// TIA Portal V19 program export: 1 tag tables, 1 data types, 3 data blocks, 18 code blocks (in call order from the OBs), 11 instance data blocks

VAR_GLOBAL   // PLC tag table "Default tag table"
   System_Byte AT %MB1 : Byte;
   FirstScan AT %M1.0 : Bool;
   DiagStatusUpdate AT %M1.1 : Bool;
   AlwaysTRUE AT %M1.2 : Bool;
   AlwaysFALSE AT %M1.3 : Bool;
   Clock_Byte AT %MB0 : Byte;
   Clock_10Hz AT %M0.0 : Bool;
   Clock_5Hz AT %M0.1 : Bool;
   "Clock_2.5Hz" AT %M0.2 : Bool;
   Clock_2Hz AT %M0.3 : Bool;
   "Clock_1.25Hz" AT %M0.4 : Bool;
   Clock_1Hz AT %M0.5 : Bool;
   "Clock_0.625Hz" AT %M0.6 : Bool;
   "Clock_0.5Hz" AT %M0.7 : Bool;
   Emergency_Stop_OK AT %M52.2 : Bool;   // Emergency status. 0 = OK, 1 = Emergency
   Emergency_Stop_Status_150K1 AT %I1.0 : Bool;   // Emergency signal from 150K1
   Sensor_102B2 AT %I1.1 : Bool;   // Sensor on conveyor - Front
   Sensor_102B3 AT %I1.2 : Bool;   // Sensor on conveyor - Middle
   Sensor_102B4 AT %I1.3 : Bool;   // Sensor on conveyor - Back
   Sensor_102B5 AT %I1.4 : Bool;   // Paint level sensor - High
   Sensor_102B6 AT %I1.5 : Bool;   // Paint level sensor - Low
   Valve_106Q6 AT %Q1.0 : Bool;   // Paint dispenser valve
   Motor_4Q3 AT %Q1.1 : Bool;   // Contactor for motor - Grinder
   Motor_4Q5 AT %Q1.2 : Bool;   // Contactor for motor - Paint
   Motor_6Q1 AT %Q1.3 : Bool;   // Contactor for motor - Ventilation
   Motor_6Q3 AT %Q1.4 : Bool;   // Contactor for motor - Vacuum
   Reset_Safety_150K1 AT %Q1.5 : Bool;   // Signal to 150K1 for emergency reset
   HMI_Start AT %M51.6 : Bool;   // HMI button signal - Start
   HMI_Pause AT %M51.7 : Bool;   // HMI button signal - Pause
   HMI_Reset AT %M52.0 : Bool;   // HMI button signal - Reset
   Input0 AT %I0.0 : Bool;
   Input1 AT %I0.1 : Bool;
   Input2 AT %I0.2 : Bool;
   Input3 AT %I0.3 : Bool;
   Input4 AT %I0.4 : Bool;
   Input5 AT %I0.5 : Bool;
   Input6 AT %I0.6 : Bool;
   Input7 AT %I0.7 : Bool;
   Input8 AT %I1.6 : Bool;
   Output0 AT %Q0.0 : Bool;
   Output1 AT %Q0.1 : Bool;
   Output2 AT %Q0.2 : Bool;
   Output3 AT %Q0.3 : Bool;
   Output4 AT %Q0.4 : Bool;
   Output5 AT %Q0.5 : Bool;
   Output6 AT %Q0.6 : Bool;
   Output7 AT %Q0.7 : Bool;
   Output8 AT %Q1.6 : Bool;
END_VAR

TYPE "XYZ_Coordinates"
   STRUCT
      X : Int;
      Y : Int;
      Z : Int;
      Mode : Int;
   END_STRUCT;
END_TYPE

DATA_BLOCK "DB_Arduino_Data"   // DB3
{ S7_Optimized_Access := 'FALSE' }
   VAR
      Read_Data : Array[1..120] of Word;
      Write_Data : Array[1..120] of Word;
   END_VAR
BEGIN
   Write_Data[1] := 16#B;
   Write_Data[2] := 16#E;
   Write_Data[3] := 16#0;
END_DATA_BLOCK

DATA_BLOCK "DB_Arduino_Tcp_Connect"   // DB10
{ S7_Optimized_Access := 'TRUE' }
// stored: MemoryReserve 100
   VAR
      MB_Arduino_Write : TCON_IP_v4;
      MB_Arduino_Read : TCON_IP_v4;
      MB_Arduino_Disconnect { S7_SetPoint := 'True'} : Bool;
      MB_Arduino_Req : Bool;
      MB_Arduino_Error : Bool;
      MB_Arduino_Done : Bool;
      MB_Arduino_Busy : Bool;
      MB_Arduino_Status : Word;
      MB_Arduino_Write_Busy : Bool;
      MB_Arduino_Write_Done : Bool;
      MB_Arduino_Write_Error : Bool;
      MB_Arduino_Write_Req : Bool;
      MB_Arduino_Write_Disconnect : Bool;
      MB_Arduino_Write_Status : Word;
   END_VAR
BEGIN
   MB_Arduino_Write.InterfaceId := 64;
   MB_Arduino_Write.ID := 16#1;
   MB_Arduino_Write.ConnectionType := 16#0B;
   MB_Arduino_Write.ActiveEstablished := 1;
   MB_Arduino_Write.RemoteAddress.ADDR[1] := 16#C0;
   MB_Arduino_Write.RemoteAddress.ADDR[2] := 16#A8;
   MB_Arduino_Write.RemoteAddress.ADDR[3] := 16#1;
   MB_Arduino_Write.RemoteAddress.ADDR[4] := 16#3D;
   MB_Arduino_Write.RemotePort := 502;
   MB_Arduino_Read.InterfaceId := 64;
   MB_Arduino_Read.ID := 16#1;
   MB_Arduino_Read.ConnectionType := 16#0B;
   MB_Arduino_Read.ActiveEstablished := 1;
   MB_Arduino_Read.RemoteAddress.ADDR[1] := 16#C0;
   MB_Arduino_Read.RemoteAddress.ADDR[2] := 16#A8;
   MB_Arduino_Read.RemoteAddress.ADDR[3] := 16#1;
   MB_Arduino_Read.RemoteAddress.ADDR[4] := 16#3D;
   MB_Arduino_Read.RemotePort := 502;
END_DATA_BLOCK

DATA_BLOCK "Letter_A"   // DB4
{ S7_Optimized_Access := 'TRUE' }
// stored: MemoryReserve 100
   VAR
      Coordinates : Array[0..5] of "XYZ_Coordinates";
   END_VAR
BEGIN
   Coordinates[0..2].X := 1.0;
   Coordinates[0..2].Y := 2.0;
   Coordinates[0..2].Z := 3.0;
END_DATA_BLOCK

ORGANIZATION_BLOCK "Main"   // OB1, LAD, ProgramCycle
TITLE = "Main Program Sweep (Cycle)"
{ S7_Optimized_Access := 'TRUE' }
// stored: SetENOAutomatically false
   VAR_INPUT
      Initial_Call : Bool;   // Initial call of this OB
      Remanence : Bool;   // =True, if remanent data are available
   END_VAR
   VAR_TEMP   // added for the SCL form of the ladder/FBD networks
      _w1 : Bool;
   END_VAR
BEGIN

REGION Network 1
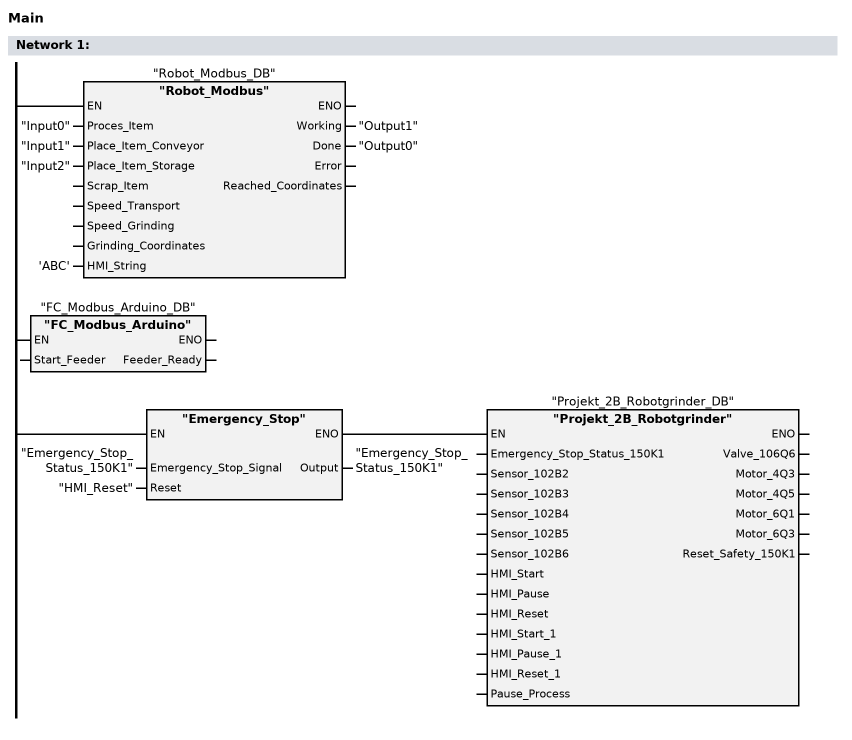
   RUNG wire#powerrail
      "Robot_Modbus_DB"(Proces_Item := "Input0", Place_Item_Conveyor := "Input1", Place_Item_Storage := "Input2", Scrap_Item :=, Speed_Transport :=, Speed_Grinding :=, Grinding_Coordinates :=, HMI_String := 'ABC', Working => "Output1", Done => "Output0", Error =>, Reached_Coordinates =>)
   END_RUNG
   RUNG wire#powerrail
      "FC_Modbus_Arduino_DB"(Start_Feeder :=, Feeder_Ready =>)
   END_RUNG
   RUNG wire#powerrail
      "Emergency_Stop"(Emergency_Stop_Signal := "Emergency_Stop_Status_150K1", Reset := "HMI_Reset", Output => "Emergency_Stop_Status_150K1")
      "Projekt_2B_Robotgrinder_DB"(Emergency_Stop_Status_150K1 :=, Sensor_102B2 :=, Sensor_102B3 :=, Sensor_102B4 :=, Sensor_102B5 :=, Sensor_102B6 :=, HMI_Start :=, HMI_Pause :=, HMI_Reset :=, HMI_Start_1 :=, HMI_Pause_1 :=, HMI_Reset_1 :=, Pause_Process :=, Valve_106Q6 =>, Motor_4Q3 =>, Motor_4Q5 =>, Motor_6Q1 =>, Motor_6Q3 =>, Reset_Safety_150K1 =>)
   END_RUNG
   // the same network as SCL:
   "Robot_Modbus_DB"(Proces_Item := "Input0",   // "Robot_Modbus"
                     Place_Item_Conveyor := "Input1",
                     Place_Item_Storage := "Input2",
                     HMI_String := 'ABC',
                     Working => "Output1",
                     Done => "Output0");
   "FC_Modbus_Arduino_DB"();   // "FC_Modbus_Arduino"
   "Emergency_Stop"(Emergency_Stop_Signal := "Emergency_Stop_Status_150K1",
                    Reset := "HMI_Reset",
                    Output => "Emergency_Stop_Status_150K1",
                    ENO => #_w1);
   IF #_w1 THEN
       "Projekt_2B_Robotgrinder_DB"();   // "Projekt_2B_Robotgrinder"
   END_IF;
END_REGION
END_ORGANIZATION_BLOCK

FUNCTION_BLOCK "Robot_Modbus"   // FB1, LAD
{ S7_Optimized_Access := 'TRUE' }
// V.0.1.1 - Updated UR robot array address
// V.0.1.0 - Created function block
// stored: MemoryReserve 100, SetENOAutomatically false
   VAR_INPUT
      Proces_Item : Bool;
      Place_Item_Conveyor : Bool;
      Place_Item_Storage : Bool;
      Scrap_Item : Bool;
      Speed_Transport : Int := 10;
      Speed_Grinding : Int := 10;
      Grinding_Coordinates : Bool;
      HMI_String : String;
   END_VAR
   VAR_OUTPUT
      Working : Bool;
      Done : Bool;
      Error : Bool;
      Reached_Coordinates : Bool;
   END_VAR
   VAR
      DISCONNECT : Bool;
      Address : TCON_IP_v4;
      Receive_Data : Int;
      Send_Data : Array[0..63] of Bool;
      Send_Coordinates : Array[0..2] of Int;
      Letter_A : Array[0..20] of "XYZ_Coordinates";
      Letter_Steps { S7_SetPoint := 'True'} : Int;
      Rising_edge : Bool;
      String_To_Letter_Array : Array[0..16] of Char;
      String_Length : Int;
      Currently_Processing : Int;
      Send_Letter_A : Bool;
      Send_Letter_B : Bool;
      Send_Letter_C : Bool;
      MB_Client_Mode : Int;
      MB_Client_Modbus_Address : Int;
      For_Loop_Counter : Int;
   END_VAR
   // Address.InterfaceId := 64;
   // Address.ID := 1;
   // Address.ConnectionType := 11;
   // Address.ActiveEstablished := TRUE;
   // Address.RemoteAddress.ADDR[1] := 192;
   // Address.RemoteAddress.ADDR[2] := 168;
   // Address.RemoteAddress.ADDR[3] := 1;
   // Address.RemoteAddress.ADDR[4] := 51;
   // Address.RemotePort := 502;
   // Address.LocalPort := 502;
   // Letter_A[0..1].X := 4;
   // Letter_A[2].X := 42;
   // Letter_A[3].X := 56;
   // Letter_A[4].X := 98;
   // Letter_A[5].X := 82;
   // Letter_A[6].X := 70;
   // Letter_A[7].X := 29;
   // Letter_A[8].X := 17;
   // Letter_A[9..10].X := 4;
   // Letter_A[11..12].X := 67;
   // Letter_A[13].X := 56;
   // Letter_A[14].X := 52;
   // Letter_A[15].X := 49;
   // Letter_A[16].X := 47;
   // Letter_A[17].X := 44;
   // Letter_A[18..19].X := 33;
   // Letter_A[0].Y := 0;
   // Letter_A[2..3].Y := 100;
   // Letter_A[4..5].Y := 0;
   // Letter_A[6..7].Y := 30;
   // Letter_A[8..10].Y := 0;
   // Letter_A[11..12].Y := 41;
   // Letter_A[13].Y := 69;
   // Letter_A[14].Y := 82;
   // Letter_A[15].Y := 90;
   // Letter_A[16].Y := 80;
   // Letter_A[17].Y := 70;
   // Letter_A[18..19].Y := 41;
   // Letter_A[1..9].Z := -1;
   // Letter_A[10].Z := 0;
   // Letter_A[12..18].Z := -1;
   // Letter_A[19].Z := 0;
   // Letter_A[14].I := 394;
   // Letter_A[15].I := 156;
   // Letter_A[16].I := -122;
   // Letter_A[17].I := -127;
   // Letter_A[14].J := 149;
   // Letter_A[15].J := 53;
   // Letter_A[16].J := 24;
   // Letter_A[17].J := 36;
   VAR_TEMP   // added for the SCL form of the ladder/FBD networks
      _w1 : Bool;
   END_VAR
BEGIN

REGION Network 1: MB_CLIENT
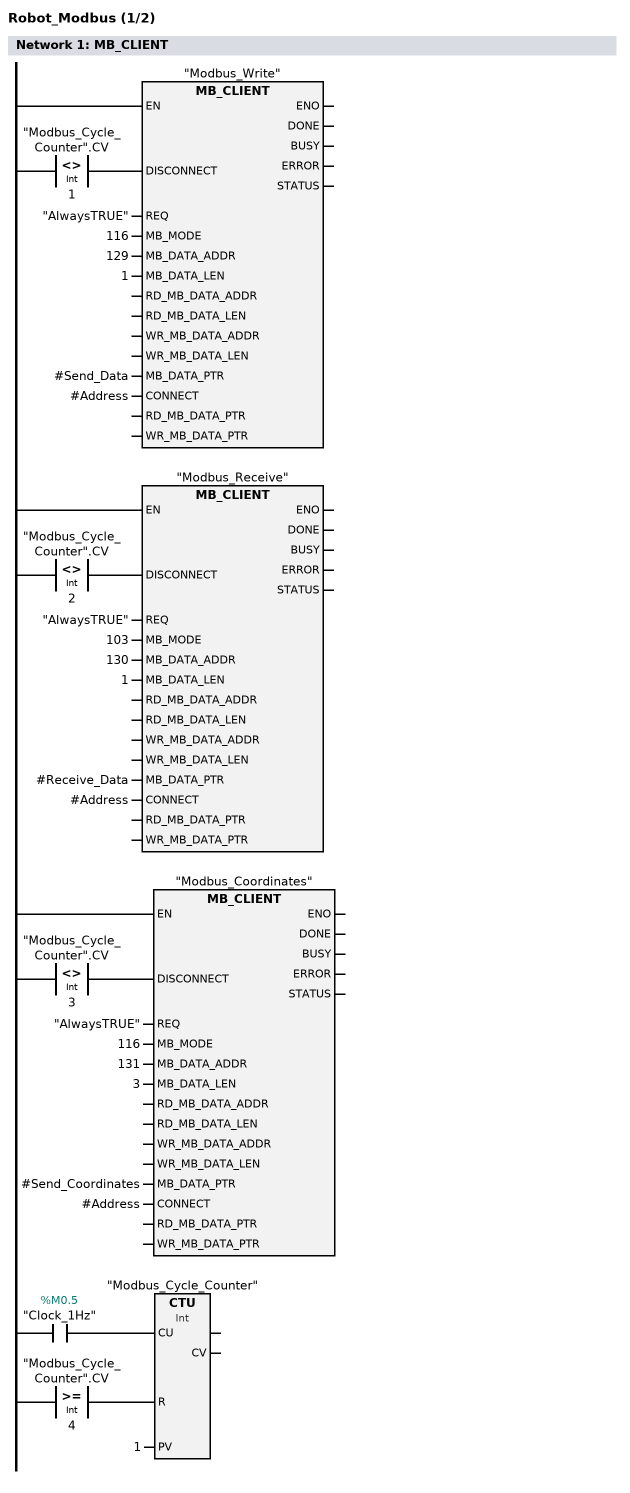
   RUNG wire#powerrail
      "Modbus_Write".MB_CLIENT(DISCONNECT := wire#w1, REQ := "AlwaysTRUE", MB_MODE := 116, MB_DATA_ADDR := 129, MB_DATA_LEN := 1, RD_MB_DATA_ADDR :=, RD_MB_DATA_LEN :=, WR_MB_DATA_ADDR :=, WR_MB_DATA_LEN :=, MB_DATA_PTR := #Send_Data, CONNECT := #Address, RD_MB_DATA_PTR :=, WR_MB_DATA_PTR :=, DONE =>, BUSY =>, ERROR =>, STATUS =>)
   END_RUNG
   RUNG wire#powerrail
      { S7_Templates := "SrcType := Int" } NE_Contact(in1 := "Modbus_Cycle_Counter".CV, in2 := 1)
   END_RUNG wire#w1
   RUNG wire#powerrail
      "Modbus_Receive".MB_CLIENT(DISCONNECT := wire#w2, REQ := "AlwaysTRUE", MB_MODE := 103, MB_DATA_ADDR := 130, MB_DATA_LEN := 1, RD_MB_DATA_ADDR :=, RD_MB_DATA_LEN :=, WR_MB_DATA_ADDR :=, WR_MB_DATA_LEN :=, MB_DATA_PTR := #Receive_Data, CONNECT := #Address, RD_MB_DATA_PTR :=, WR_MB_DATA_PTR :=, DONE =>, BUSY =>, ERROR =>, STATUS =>)
   END_RUNG
   RUNG wire#powerrail
      { S7_Templates := "SrcType := Int" } NE_Contact(in1 := "Modbus_Cycle_Counter".CV, in2 := 2)
   END_RUNG wire#w2
   RUNG wire#powerrail
      "Modbus_Coordinates".MB_CLIENT(DISCONNECT := wire#w3, REQ := "AlwaysTRUE", MB_MODE := 116, MB_DATA_ADDR := 131, MB_DATA_LEN := 3, RD_MB_DATA_ADDR :=, RD_MB_DATA_LEN :=, WR_MB_DATA_ADDR :=, WR_MB_DATA_LEN :=, MB_DATA_PTR := #Send_Coordinates, CONNECT := #Address, RD_MB_DATA_PTR :=, WR_MB_DATA_PTR :=, DONE =>, BUSY =>, ERROR =>, STATUS =>)
   END_RUNG
   RUNG wire#powerrail
      { S7_Templates := "SrcType := Int" } NE_Contact(in1 := "Modbus_Cycle_Counter".CV, in2 := 3)
   END_RUNG wire#w3
   RUNG wire#powerrail
      Contact( "Clock_1Hz" )
      { S7_Templates := "value_type := Int" } "Modbus_Cycle_Counter".CTU(r := wire#w4, pv := 1, cv =>)
   END_RUNG
   RUNG wire#powerrail
      { S7_Templates := "SrcType := Int" } GE_Contact(in1 := "Modbus_Cycle_Counter".CV, in2 := 4)
   END_RUNG wire#w4
   // the same network as SCL:
   "Modbus_Write"(DISCONNECT := "Modbus_Cycle_Counter".CV <> 1,   // MB_CLIENT
                  REQ := "AlwaysTRUE",
                  MB_MODE := 116,
                  MB_DATA_ADDR := 129,
                  MB_DATA_LEN := 1,
                  MB_DATA_PTR := #Send_Data,
                  CONNECT := #Address);
   "Modbus_Receive"(DISCONNECT := "Modbus_Cycle_Counter".CV <> 2,   // MB_CLIENT
                    REQ := "AlwaysTRUE",
                    MB_MODE := 103,
                    MB_DATA_ADDR := 130,
                    MB_DATA_LEN := 1,
                    MB_DATA_PTR := #Receive_Data,
                    CONNECT := #Address);
   "Modbus_Coordinates"(DISCONNECT := "Modbus_Cycle_Counter".CV <> 3,   // MB_CLIENT
                        REQ := "AlwaysTRUE",
                        MB_MODE := 116,
                        MB_DATA_ADDR := 131,
                        MB_DATA_LEN := 3,
                        MB_DATA_PTR := #Send_Coordinates,
                        CONNECT := #Address);
   "Modbus_Cycle_Counter".CTU(CU := "Clock_1Hz", R := "Modbus_Cycle_Counter".CV >= 4, PV := 1);
END_REGION

REGION Network 2: Send Data
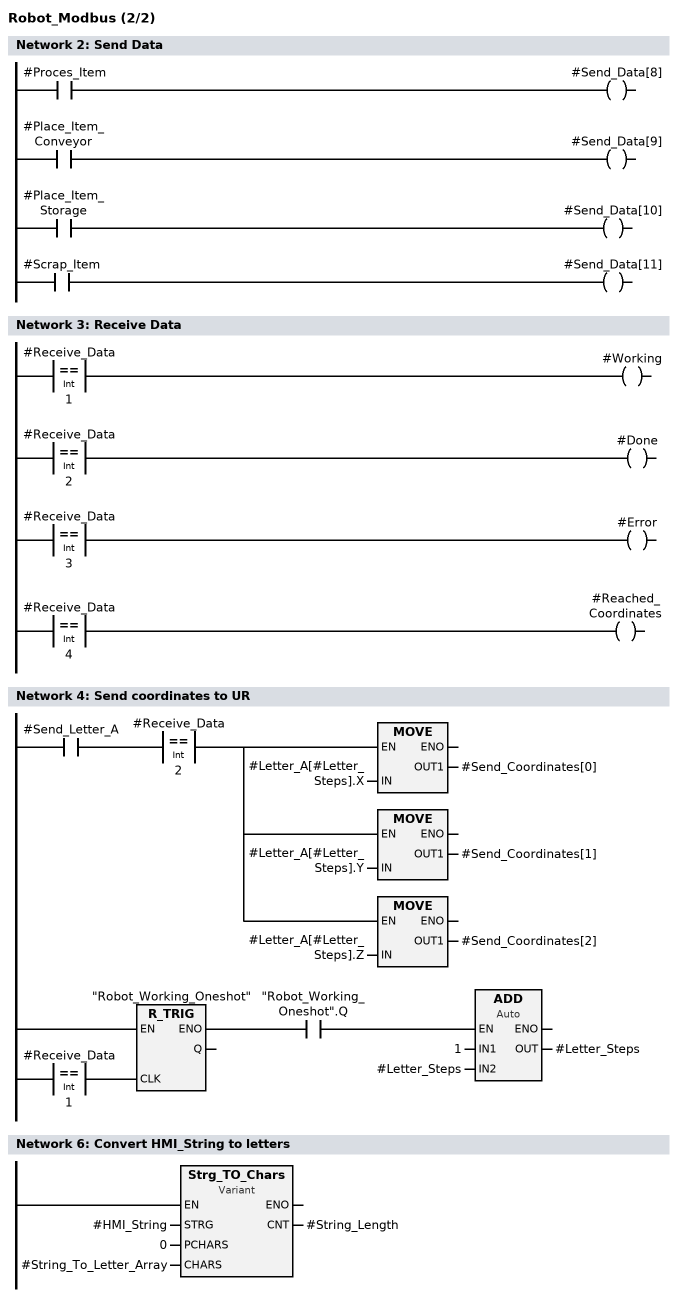
   RUNG wire#powerrail
      Contact( #Proces_Item )
      Coil( #Send_Data[8] )
   END_RUNG
   RUNG wire#powerrail
      Contact( #Place_Item_Conveyor )
      Coil( #Send_Data[9] )
   END_RUNG
   RUNG wire#powerrail
      Contact( #Place_Item_Storage )
      Coil( #Send_Data[10] )
   END_RUNG
   RUNG wire#powerrail
      Contact( #Scrap_Item )
      Coil( #Send_Data[11] )
   END_RUNG
   // the same network as SCL:
   #Send_Data[8] := #Proces_Item;
   #Send_Data[9] := #Place_Item_Conveyor;
   #Send_Data[10] := #Place_Item_Storage;
   #Send_Data[11] := #Scrap_Item;
END_REGION

REGION Network 3: Receive Data
   RUNG wire#powerrail
      { S7_Templates := "SrcType := Int" } EQ_Contact(in1 := #Receive_Data, in2 := 1)
      Coil( #Working )
   END_RUNG
   RUNG wire#powerrail
      { S7_Templates := "SrcType := Int" } EQ_Contact(in1 := #Receive_Data, in2 := 2)
      Coil( #Done )
   END_RUNG
   RUNG wire#powerrail
      { S7_Templates := "SrcType := Int" } EQ_Contact(in1 := #Receive_Data, in2 := 3)
      Coil( #Error )
   END_RUNG
   RUNG wire#powerrail
      { S7_Templates := "SrcType := Int" } EQ_Contact(in1 := #Receive_Data, in2 := 4)
      Coil( #Reached_Coordinates )
   END_RUNG
   // the same network as SCL:
   #Working := #Receive_Data = 1;
   #Done := #Receive_Data = 2;
   #Error := #Receive_Data = 3;
   #Reached_Coordinates := #Receive_Data = 4;
END_REGION

REGION Network 4: Send coordinates to UR
   RUNG wire#powerrail
      Contact( #Send_Letter_A )
      { S7_Templates := "SrcType := Int" } EQ_Contact(in1 := #Receive_Data, in2 := 2)
      wire#w1
      Move(in := #Letter_A[#Letter_Steps].X, out1 => #Send_Coordinates[0])
   END_RUNG
   RUNG wire#w1
      Move(in := #Letter_A[#Letter_Steps].Y, out1 => #Send_Coordinates[1])
   END_RUNG
   RUNG wire#w1
      Move(in := #Letter_A[#Letter_Steps].Z, out1 => #Send_Coordinates[2])
   END_RUNG
   RUNG wire#powerrail
      "Robot_Working_Oneshot".R_TRIG(CLK := wire#w2, Q =>)
      Contact( "Robot_Working_Oneshot".Q )
      Add(in1 := 1, in2 := #Letter_Steps, out => #Letter_Steps)
   END_RUNG
   RUNG wire#powerrail
      { S7_Templates := "SrcType := Int" } EQ_Contact(in1 := #Receive_Data, in2 := 1)
   END_RUNG wire#w2
   // the same network as SCL:
   IF #Send_Letter_A AND (#Receive_Data = 2) THEN
       #Send_Coordinates[0] := #Letter_A[#Letter_Steps].X;
       #Send_Coordinates[1] := #Letter_A[#Letter_Steps].Y;
       #Send_Coordinates[2] := #Letter_A[#Letter_Steps].Z;
   END_IF;
   "Robot_Working_Oneshot"(CLK := #Receive_Data = 1, ENO => #_w1);   // R_TRIG
   IF #_w1 AND "Robot_Working_Oneshot".Q THEN #Letter_Steps := 1 + #Letter_Steps; END_IF;
END_REGION

REGION Network 5 (SCL): Insert coordinates into Modbus_Data array
   (*
   //If we need to make letter A, and robot is sending ready signal
   IF #Send_Letter_A AND #Send_Data[25] THEN

       FOR #For_Loop_Counter := 32 TO 48 DO
           //Find the bit state inside to INT of letter_A array, and copy that to the Modbus data array
           //The for loop repeats the steps again for the array posistions 32-48
           #Letter_A[#Letter_Steps].X.%X0 := #Send_Data[#For_Loop_Counter];
       END_FOR;

       FOR #For_Loop_Counter := 49 TO 64 DO
           #Letter_A[#Letter_Steps].Y.%X0 := #Send_Data[#For_Loop_Counter];
       END_FOR;

       FOR #For_Loop_Counter := 65 TO 79 DO
           #Letter_A[#Letter_Steps].Z.%X0 := #Send_Data[#For_Loop_Counter];
       END_FOR;

   END_IF; *)
END_REGION

REGION Network 6: Convert HMI_String to letters
   RUNG wire#powerrail
      { S7_Templates := "[ptr_type := Variant, strg_type := String]" } Strg_TO_Chars(Strg := #HMI_String, pChars := 0, Chars := #String_To_Letter_Array, Cnt => #String_Length)
   END_RUNG
   // the same network as SCL:
   Strg_TO_Chars(Strg := #HMI_String, pChars := 0, Chars := #String_To_Letter_Array, Cnt => #String_Length);
END_REGION

REGION Network 7 (SCL)
   IF #Currently_Processing < #String_Length THEN //Hvis vi ikke er nået forbi enden af teksten

       IF #String_To_Letter_Array[#Currently_Processing] = 'A' THEN //Hvis der på position X, er et "A" i teksten
           #Send_Letter_A := TRUE;
       ELSIF #String_To_Letter_Array[#Currently_Processing] = 'B' THEN
           #Send_Letter_B := TRUE;
       ELSIF #String_To_Letter_Array[#Currently_Processing] = 'C' THEN
           #Send_Letter_B := TRUE;
       END_IF;
   END_IF;
END_REGION
END_FUNCTION_BLOCK

FUNCTION_BLOCK "FC_Modbus_Arduino"   // FB1, LAD
{ S7_Optimized_Access := 'TRUE' }
// stored: MemoryReserve 100, SetENOAutomatically false
   VAR_INPUT
      Start_Feeder : Bool;
   END_VAR
   VAR_OUTPUT
      Feeder_Ready : Bool;
   END_VAR
BEGIN

REGION Network 1
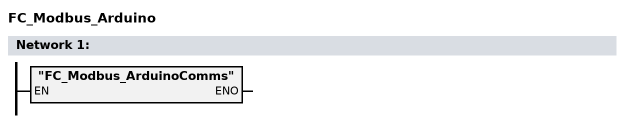
   RUNG wire#powerrail
      "FC_Modbus_ArduinoComms"()
   END_RUNG
   // the same network as SCL:
   "FC_Modbus_ArduinoComms"();
END_REGION
END_FUNCTION_BLOCK

FUNCTION "FC_Modbus_ArduinoComms" : Void   // FC1, LAD
{ S7_Optimized_Access := 'TRUE' }
// stored: SetENOAutomatically false
BEGIN

REGION Network 1
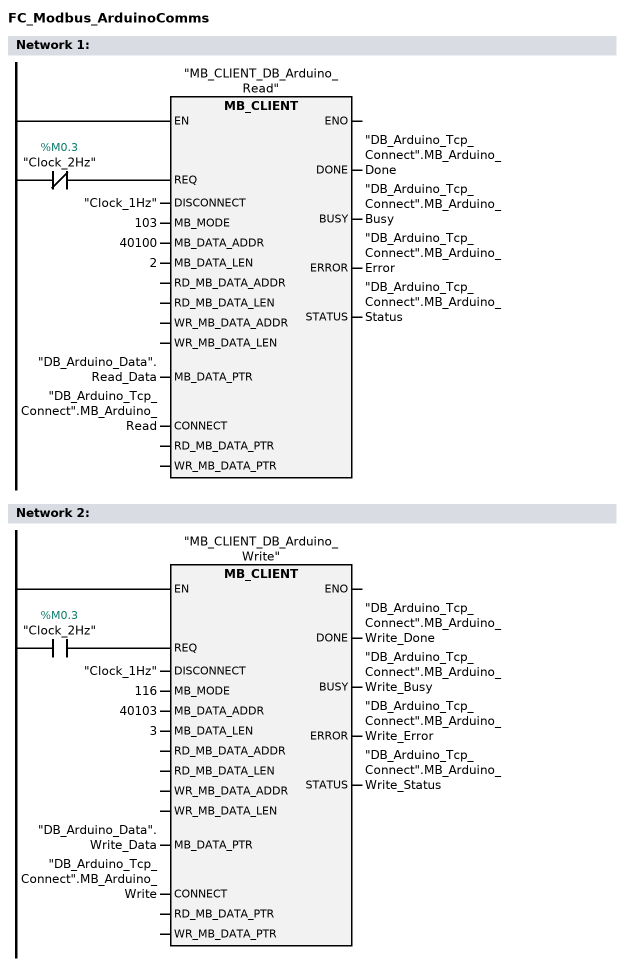
   RUNG wire#powerrail
      "MB_CLIENT_DB_Arduino_Read".MB_CLIENT(REQ := wire#w1, DISCONNECT := "Clock_1Hz", MB_MODE := 103, MB_DATA_ADDR := 40100, MB_DATA_LEN := 2, RD_MB_DATA_ADDR :=, RD_MB_DATA_LEN :=, WR_MB_DATA_ADDR :=, WR_MB_DATA_LEN :=, MB_DATA_PTR := "DB_Arduino_Data".Read_Data, CONNECT := "DB_Arduino_Tcp_Connect".MB_Arduino_Read, RD_MB_DATA_PTR :=, WR_MB_DATA_PTR :=, DONE => "DB_Arduino_Tcp_Connect".MB_Arduino_Done, BUSY => "DB_Arduino_Tcp_Connect".MB_Arduino_Busy, ERROR => "DB_Arduino_Tcp_Connect".MB_Arduino_Error, STATUS => "DB_Arduino_Tcp_Connect".MB_Arduino_Status)
   END_RUNG
   RUNG wire#powerrail
      I_Contact( "Clock_2Hz" )
   END_RUNG wire#w1
   // the same network as SCL:
   "MB_CLIENT_DB_Arduino_Read"(REQ := NOT "Clock_2Hz",   // MB_CLIENT
                           DISCONNECT := "Clock_1Hz",
                           MB_MODE := 103,
                           MB_DATA_ADDR := 40100,
                           MB_DATA_LEN := 2,
                           MB_DATA_PTR := "DB_Arduino_Data".Read_Data,
                           CONNECT := "DB_Arduino_Tcp_Connect".MB_Arduino_Read,
                           DONE => "DB_Arduino_Tcp_Connect".MB_Arduino_Done,
                           BUSY => "DB_Arduino_Tcp_Connect".MB_Arduino_Busy,
                           ERROR => "DB_Arduino_Tcp_Connect".MB_Arduino_Error,
                           STATUS => "DB_Arduino_Tcp_Connect".MB_Arduino_Status);
END_REGION

REGION Network 2
   RUNG wire#powerrail
      "MB_CLIENT_DB_Arduino_Write".MB_CLIENT(REQ := wire#w1, DISCONNECT := "Clock_1Hz", MB_MODE := 116, MB_DATA_ADDR := 40103, MB_DATA_LEN := 3, RD_MB_DATA_ADDR :=, RD_MB_DATA_LEN :=, WR_MB_DATA_ADDR :=, WR_MB_DATA_LEN :=, MB_DATA_PTR := "DB_Arduino_Data".Write_Data, CONNECT := "DB_Arduino_Tcp_Connect".MB_Arduino_Write, RD_MB_DATA_PTR :=, WR_MB_DATA_PTR :=, DONE => "DB_Arduino_Tcp_Connect".MB_Arduino_Write_Done, BUSY => "DB_Arduino_Tcp_Connect".MB_Arduino_Write_Busy, ERROR => "DB_Arduino_Tcp_Connect".MB_Arduino_Write_Error, STATUS => "DB_Arduino_Tcp_Connect".MB_Arduino_Write_Status)
   END_RUNG
   RUNG wire#powerrail
      Contact( "Clock_2Hz" )
   END_RUNG wire#w1
   // the same network as SCL:
   "MB_CLIENT_DB_Arduino_Write"(REQ := "Clock_2Hz",   // MB_CLIENT
                           DISCONNECT := "Clock_1Hz",
                           MB_MODE := 116,
                           MB_DATA_ADDR := 40103,
                           MB_DATA_LEN := 3,
                           MB_DATA_PTR := "DB_Arduino_Data".Write_Data,
                           CONNECT := "DB_Arduino_Tcp_Connect".MB_Arduino_Write,
                           DONE => "DB_Arduino_Tcp_Connect".MB_Arduino_Write_Done,
                           BUSY => "DB_Arduino_Tcp_Connect".MB_Arduino_Write_Busy,
                           ERROR => "DB_Arduino_Tcp_Connect".MB_Arduino_Write_Error,
                           STATUS => "DB_Arduino_Tcp_Connect".MB_Arduino_Write_Status);
END_REGION
END_FUNCTION

FUNCTION "Emergency_Stop" : Void
{ S7_Optimized_Access := 'TRUE' }
VERSION : 0.1
   VAR_INPUT 
      Emergency_Stop_Signal : Bool;
      Reset : Bool;
   END_VAR

   VAR_OUTPUT 
      Output : Bool;
   END_VAR


BEGIN
	IF #Emergency_Stop_Signal = TRUE THEN
	    #Output := TRUE;
	END_IF;
	    
	IF #Reset = TRUE AND #Emergency_Stop_Signal = FALSE THEN
	    #Output := FALSE;
	END_IF;
END_FUNCTION

FUNCTION_BLOCK "Projekt_2B_Robotgrinder"   // FB4, LAD
{ S7_Optimized_Access := 'TRUE' }
// stored: MemoryReserve 100, SetENOAutomatically false
   VAR_INPUT
      Emergency_Stop_Status_150K1 : Bool;
      Sensor_102B2 : Bool;
      Sensor_102B3 : Bool;
      Sensor_102B4 : Bool;
      Sensor_102B5 : Bool;
      Sensor_102B6 : Bool;
      HMI_Start : Bool;
      HMI_Pause : Bool;
      HMI_Reset : Bool;
      HMI_Start_1 : Bool;
      HMI_Pause_1 : Bool;
      HMI_Reset_1 : Bool;
      Pause_Process : Bool;
   END_VAR
   VAR_OUTPUT
      Valve_106Q6 : Bool;
      Motor_4Q3 : Bool;
      Motor_4Q5 : Bool;
      Motor_6Q1 : Bool;
      Motor_6Q3 : Bool;
      Reset_Safety_150K1 : Bool;
   END_VAR
   VAR
      Main_Step : Int;
      Process_Step : Int;
      Reset_Step : Int;
      Placement_Step : Int;
      Order_Amount : Int;
      Items_Produced : Int;
      Items_Delivered : Int;
      Total_orders : Int;
      Storage_Amount : Int;
      Storage_Plus_Produce : Int;
      Storage_Min : Int;
      Storage_Max : Int;
      Robot_Done : Bool;
   END_VAR
BEGIN

REGION Network 1: Main Process Step 0
   // If the system is currently idling, then pressing start will start the process. On PLC restart, moves starting values into steps.
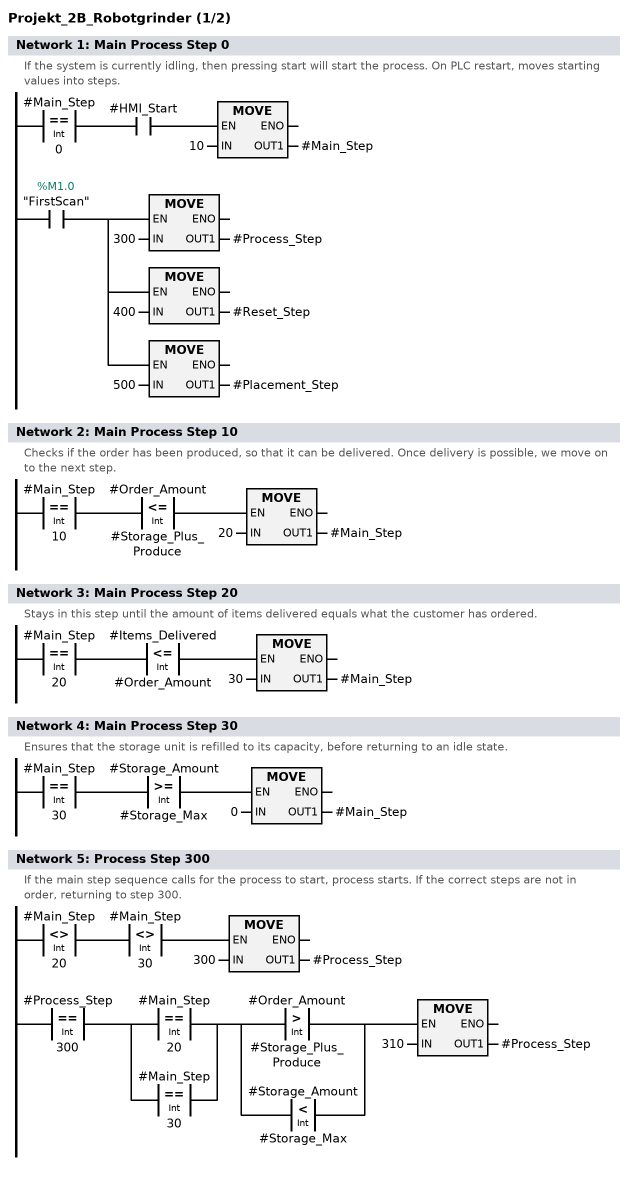
   RUNG wire#powerrail
      { S7_Templates := "SrcType := Int" } EQ_Contact(in1 := #Main_Step, in2 := 0)
      Contact( #HMI_Start )
      Move(in := 10, out1 => #Main_Step)
   END_RUNG
   RUNG wire#powerrail
      Contact( "FirstScan" )
      wire#w1
      Move(in := 300, out1 => #Process_Step)
   END_RUNG
   RUNG wire#w1
      Move(in := 400, out1 => #Reset_Step)
   END_RUNG
   RUNG wire#w1
      Move(in := 500, out1 => #Placement_Step)
   END_RUNG
   // the same network as SCL:
   IF (#Main_Step = 0) AND #HMI_Start THEN #Main_Step := 10; END_IF;
   IF "FirstScan" THEN
       #Process_Step := 300;
       #Reset_Step := 400;
       #Placement_Step := 500;
   END_IF;
END_REGION

REGION Network 2: Main Process Step 10
   // Checks if the order has been produced, so that it can be delivered. Once delivery is possible, we move on to the next step.
   RUNG wire#powerrail
      { S7_Templates := "SrcType := Int" } EQ_Contact(in1 := #Main_Step, in2 := 10)
      { S7_Templates := "SrcType := Int" } LE_Contact(in1 := #Order_Amount, in2 := #Storage_Plus_Produce)
      Move(in := 20, out1 => #Main_Step)
   END_RUNG
   // the same network as SCL:
   IF (#Main_Step = 10) AND (#Order_Amount <= #Storage_Plus_Produce) THEN #Main_Step := 20; END_IF;
END_REGION

REGION Network 3: Main Process Step 20
   // Stays in this step until the amount of items delivered equals what the customer has ordered.
   RUNG wire#powerrail
      { S7_Templates := "SrcType := Int" } EQ_Contact(in1 := #Main_Step, in2 := 20)
      { S7_Templates := "SrcType := Int" } LE_Contact(in1 := #Items_Delivered, in2 := #Order_Amount)
      Move(in := 30, out1 => #Main_Step)
   END_RUNG
   // the same network as SCL:
   IF (#Main_Step = 20) AND (#Items_Delivered <= #Order_Amount) THEN #Main_Step := 30; END_IF;
END_REGION

REGION Network 4: Main Process Step 30
   // Ensures that the storage unit is refilled to its capacity, before returning to an idle state.
   RUNG wire#powerrail
      { S7_Templates := "SrcType := Int" } EQ_Contact(in1 := #Main_Step, in2 := 30)
      { S7_Templates := "SrcType := Int" } GE_Contact(in1 := #Storage_Amount, in2 := #Storage_Max)
      Move(in := 0, out1 => #Main_Step)
   END_RUNG
   // the same network as SCL:
   IF (#Main_Step = 30) AND (#Storage_Amount >= #Storage_Max) THEN #Main_Step := 0; END_IF;
END_REGION

REGION Network 5: Process Step 300
   // If the main step sequence calls for the process to start, process starts. If the correct steps are not in order, returning to step 300.
   RUNG wire#powerrail
      { S7_Templates := "SrcType := Int" } NE_Contact(in1 := #Main_Step, in2 := 20)
      { S7_Templates := "SrcType := Int" } NE_Contact(in1 := #Main_Step, in2 := 30)
      Move(in := 300, out1 => #Process_Step)
   END_RUNG
   RUNG wire#powerrail
      { S7_Templates := "SrcType := Int" } EQ_Contact(in1 := #Process_Step, in2 := 300)
      wire#w1
      { S7_Templates := "SrcType := Int" } EQ_Contact(in1 := #Main_Step, in2 := 20)
      wire#w2
      { S7_Templates := "SrcType := Int" } GT_Contact(in1 := #Order_Amount, in2 := #Storage_Plus_Produce)
      wire#w3
      Move(in := 310, out1 => #Process_Step)
   END_RUNG
   RUNG wire#w1
      { S7_Templates := "SrcType := Int" } EQ_Contact(in1 := #Main_Step, in2 := 30)
   END_RUNG wire#w2
   RUNG wire#w2
      { S7_Templates := "SrcType := Int" } LT_Contact(in1 := #Storage_Amount, in2 := #Storage_Max)
   END_RUNG wire#w3
   // the same network as SCL:
   IF (#Main_Step <> 20) AND (#Main_Step <> 30) THEN #Process_Step := 300; END_IF;
   IF (#Process_Step = 300) AND ((#Main_Step = 20) OR (#Main_Step = 30)) AND ((#Order_Amount > #Storage_Plus_Produce) OR (#Storage_Amount < #Storage_Max)) THEN
       #Process_Step := 310;
   END_IF;
END_REGION

REGION Network 6: Process Step 310
   // Feeder activates in step 310. Once sensor activates by item on conveyor, moving to next step.
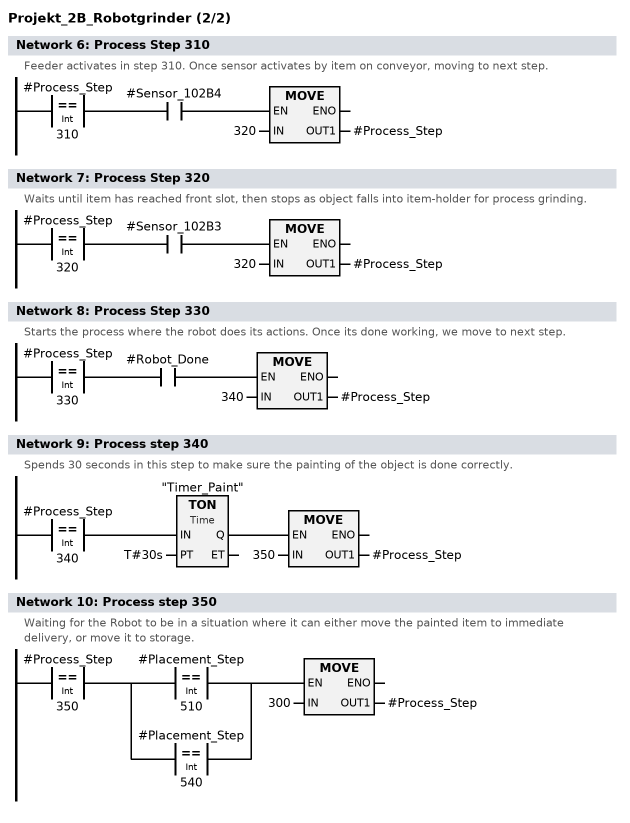
   RUNG wire#powerrail
      { S7_Templates := "SrcType := Int" } EQ_Contact(in1 := #Process_Step, in2 := 310)
      Contact( #Sensor_102B4 )
      Move(in := 320, out1 => #Process_Step)
   END_RUNG
   // the same network as SCL:
   IF (#Process_Step = 310) AND #Sensor_102B4 THEN #Process_Step := 320; END_IF;
END_REGION

REGION Network 7: Process Step 320
   // Waits until item has reached front slot, then stops as object falls into item-holder for process grinding.
   RUNG wire#powerrail
      { S7_Templates := "SrcType := Int" } EQ_Contact(in1 := #Process_Step, in2 := 320)
      Contact( #Sensor_102B3 )
      Move(in := 320, out1 => #Process_Step)
   END_RUNG
   // the same network as SCL:
   IF (#Process_Step = 320) AND #Sensor_102B3 THEN #Process_Step := 320; END_IF;
END_REGION

REGION Network 8: Process Step 330
   // Starts the process where the robot does its actions. Once its done working, we move to next step.
   RUNG wire#powerrail
      { S7_Templates := "SrcType := Int" } EQ_Contact(in1 := #Process_Step, in2 := 330)
      Contact( #Robot_Done )
      Move(in := 340, out1 => #Process_Step)
   END_RUNG
   // the same network as SCL:
   IF (#Process_Step = 330) AND #Robot_Done THEN #Process_Step := 340; END_IF;
END_REGION

REGION Network 9: Process step 340
   // Spends 30 seconds in this step to make sure the painting of the object is done correctly.
   RUNG wire#powerrail
      { S7_Templates := "SrcType := Int" } EQ_Contact(in1 := #Process_Step, in2 := 340)
      { S7_Templates := "time_type := Time" } "Timer_Paint".TON(pt := T#30s, et =>)
      Move(in := 350, out1 => #Process_Step)
   END_RUNG
   // the same network as SCL:
   "Timer_Paint".TON(IN := #Process_Step = 340, PT := T#30s);
   IF "Timer_Paint".Q THEN #Process_Step := 350; END_IF;
END_REGION

REGION Network 10: Process step 350
   // Waiting for the Robot to be in a situation where it can either move the painted item to immediate delivery, or move it to storage.
   RUNG wire#powerrail
      { S7_Templates := "SrcType := Int" } EQ_Contact(in1 := #Process_Step, in2 := 350)
      wire#w1
      { S7_Templates := "SrcType := Int" } EQ_Contact(in1 := #Placement_Step, in2 := 510)
      wire#w2
      Move(in := 300, out1 => #Process_Step)
   END_RUNG
   RUNG wire#w1
      { S7_Templates := "SrcType := Int" } EQ_Contact(in1 := #Placement_Step, in2 := 540)
   END_RUNG wire#w2
   // the same network as SCL:
   IF (#Process_Step = 350) AND ((#Placement_Step = 510) OR (#Placement_Step = 540)) THEN
       #Process_Step := 300;
   END_IF;
END_REGION
END_FUNCTION_BLOCK

ORGANIZATION_BLOCK "test"   // OB123, LAD, ProgramCycle
TITLE = "Main Program Sweep (Cycle)"
{ S7_Optimized_Access := 'TRUE' }
// stored: SetENOAutomatically false
   VAR_INPUT
      Initial_Call : Bool;   // Initial call of this OB
      Remanence : Bool;   // =True, if remanent data are available
   END_VAR
BEGIN
END_ORGANIZATION_BLOCK

FUNCTION_BLOCK "Arduino_Modbus"   // FB6, LAD
{ S7_Optimized_Access := 'TRUE' }
// v0.0.1 has not been tested
// stored: MemoryReserve 100, SetENOAutomatically false
   VAR_INPUT
      Proces_Item : Bool;
      Place_Item_Conveyor : Bool;
      Place_Item_Storage : Bool;
      Scrap_Item : Bool;
      Speed_Transport : Int := 10;
      Speed_Grinding : Int := 10;
      Grinding_Coordinates : Bool;
      Letter : DB_ANY;
   END_VAR
   VAR_OUTPUT
      Working : Bool;
      Done : Bool;
      Error : Bool;
      Reached_Coordinates : Bool;
   END_VAR
   VAR
      DISCONNECT : Bool;
      Address : TCON_IP_v4;
      ReceiveData : Array[0..5] of Int;
      SendData : Array[0..5] of Int;
   END_VAR
   // Address.InterfaceId := 64;
   // Address.ID := 1;
   // Address.ConnectionType := 11;
   // Address.ActiveEstablished := TRUE;
   // Address.RemoteAddress.ADDR[1] := 192;
   // Address.RemoteAddress.ADDR[2] := 168;
   // Address.RemoteAddress.ADDR[3] := 1;
   // Address.RemoteAddress.ADDR[4] := 61;
   // Address.RemotePort := 502;
   // Address.LocalPort := 502;
BEGIN

REGION Network 1: MB_CLIENT
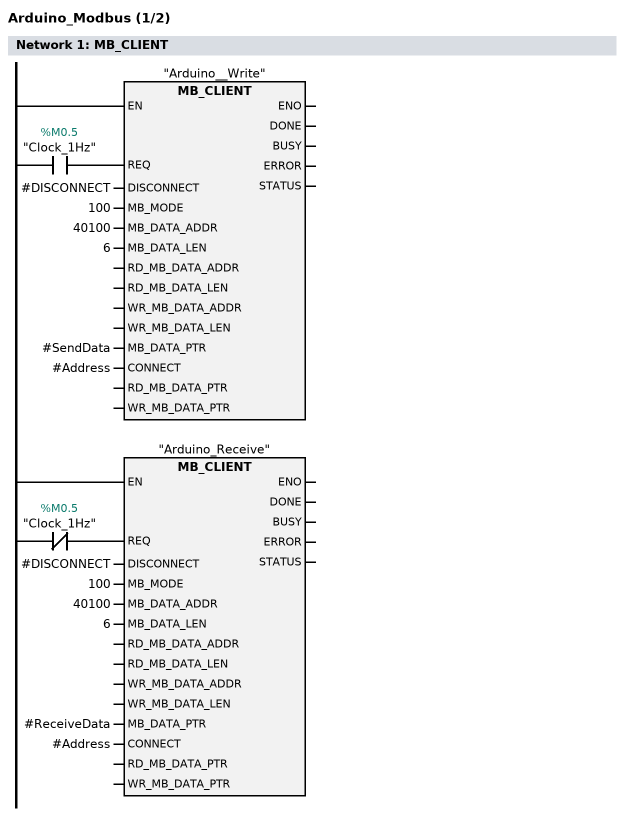
   RUNG wire#powerrail
      "Arduino__Write".MB_CLIENT(REQ := wire#w1, DISCONNECT := #DISCONNECT, MB_MODE := 100, MB_DATA_ADDR := 40100, MB_DATA_LEN := 6, RD_MB_DATA_ADDR :=, RD_MB_DATA_LEN :=, WR_MB_DATA_ADDR :=, WR_MB_DATA_LEN :=, MB_DATA_PTR := #SendData, CONNECT := #Address, RD_MB_DATA_PTR :=, WR_MB_DATA_PTR :=, DONE =>, BUSY =>, ERROR =>, STATUS =>)
   END_RUNG
   RUNG wire#powerrail
      Contact( "Clock_1Hz" )
   END_RUNG wire#w1
   RUNG wire#powerrail
      "Arduino_Receive".MB_CLIENT(REQ := wire#w2, DISCONNECT := #DISCONNECT, MB_MODE := 100, MB_DATA_ADDR := 40100, MB_DATA_LEN := 6, RD_MB_DATA_ADDR :=, RD_MB_DATA_LEN :=, WR_MB_DATA_ADDR :=, WR_MB_DATA_LEN :=, MB_DATA_PTR := #ReceiveData, CONNECT := #Address, RD_MB_DATA_PTR :=, WR_MB_DATA_PTR :=, DONE =>, BUSY =>, ERROR =>, STATUS =>)
   END_RUNG
   RUNG wire#powerrail
      I_Contact( "Clock_1Hz" )
   END_RUNG wire#w2
   // the same network as SCL:
   "Arduino__Write"(REQ := "Clock_1Hz",   // MB_CLIENT
                    DISCONNECT := #DISCONNECT,
                    MB_MODE := 100,
                    MB_DATA_ADDR := 40100,
                    MB_DATA_LEN := 6,
                    MB_DATA_PTR := #SendData,
                    CONNECT := #Address);
   "Arduino_Receive"(REQ := NOT "Clock_1Hz",   // MB_CLIENT
                     DISCONNECT := #DISCONNECT,
                     MB_MODE := 100,
                     MB_DATA_ADDR := 40100,
                     MB_DATA_LEN := 6,
                     MB_DATA_PTR := #ReceiveData,
                     CONNECT := #Address);
END_REGION

REGION Network 2: Send Data
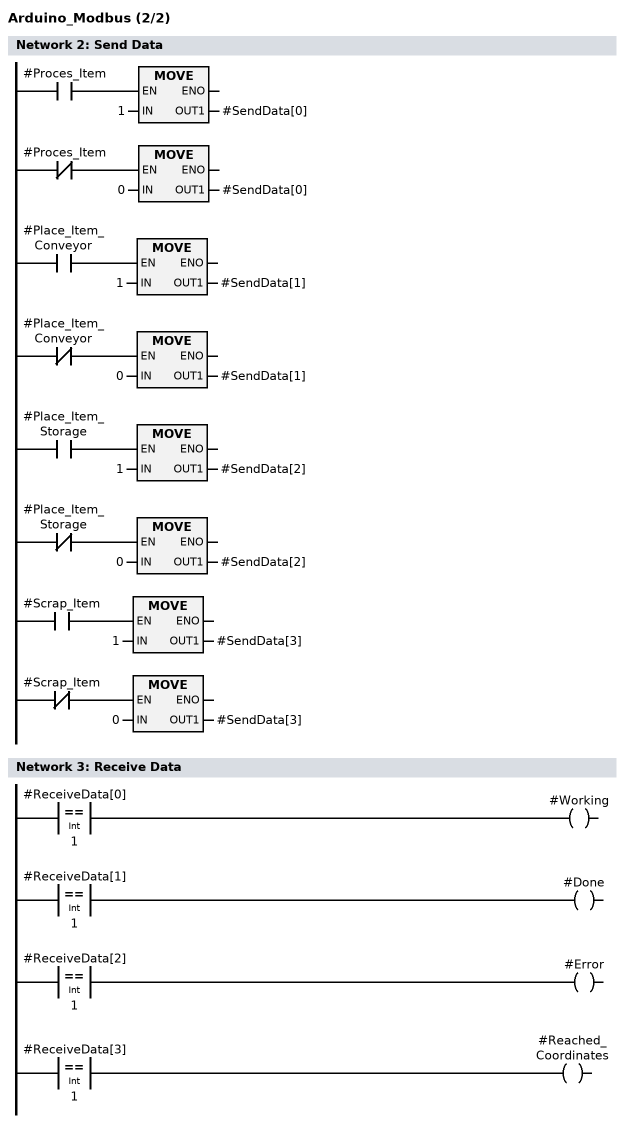
   RUNG wire#powerrail
      Contact( #Proces_Item )
      Move(in := 1, out1 => #SendData[0])
   END_RUNG
   RUNG wire#powerrail
      I_Contact( #Proces_Item )
      Move(in := 0, out1 => #SendData[0])
   END_RUNG
   RUNG wire#powerrail
      Contact( #Place_Item_Conveyor )
      Move(in := 1, out1 => #SendData[1])
   END_RUNG
   RUNG wire#powerrail
      I_Contact( #Place_Item_Conveyor )
      Move(in := 0, out1 => #SendData[1])
   END_RUNG
   RUNG wire#powerrail
      Contact( #Place_Item_Storage )
      Move(in := 1, out1 => #SendData[2])
   END_RUNG
   RUNG wire#powerrail
      I_Contact( #Place_Item_Storage )
      Move(in := 0, out1 => #SendData[2])
   END_RUNG
   RUNG wire#powerrail
      Contact( #Scrap_Item )
      Move(in := 1, out1 => #SendData[3])
   END_RUNG
   RUNG wire#powerrail
      I_Contact( #Scrap_Item )
      Move(in := 0, out1 => #SendData[3])
   END_RUNG
   // the same network as SCL:
   IF #Proces_Item THEN #SendData[0] := 1; END_IF;
   IF NOT #Proces_Item THEN #SendData[0] := 0; END_IF;
   IF #Place_Item_Conveyor THEN #SendData[1] := 1; END_IF;
   IF NOT #Place_Item_Conveyor THEN #SendData[1] := 0; END_IF;
   IF #Place_Item_Storage THEN #SendData[2] := 1; END_IF;
   IF NOT #Place_Item_Storage THEN #SendData[2] := 0; END_IF;
   IF #Scrap_Item THEN #SendData[3] := 1; END_IF;
   IF NOT #Scrap_Item THEN #SendData[3] := 0; END_IF;
END_REGION

REGION Network 3: Receive Data
   RUNG wire#powerrail
      { S7_Templates := "SrcType := Int" } EQ_Contact(in1 := #ReceiveData[0], in2 := 1)
      Coil( #Working )
   END_RUNG
   RUNG wire#powerrail
      { S7_Templates := "SrcType := Int" } EQ_Contact(in1 := #ReceiveData[1], in2 := 1)
      Coil( #Done )
   END_RUNG
   RUNG wire#powerrail
      { S7_Templates := "SrcType := Int" } EQ_Contact(in1 := #ReceiveData[2], in2 := 1)
      Coil( #Error )
   END_RUNG
   RUNG wire#powerrail
      { S7_Templates := "SrcType := Int" } EQ_Contact(in1 := #ReceiveData[3], in2 := 1)
      Coil( #Reached_Coordinates )
   END_RUNG
   // the same network as SCL:
   #Working := #ReceiveData[0] = 1;
   #Done := #ReceiveData[1] = 1;
   #Error := #ReceiveData[2] = 1;
   #Reached_Coordinates := #ReceiveData[3] = 1;
END_REGION
END_FUNCTION_BLOCK

FUNCTION_BLOCK "Painting_Chamber"   // FB4, LAD
{ S7_Optimized_Access := 'TRUE' }
// stored: MemoryReserve 100, SetENOAutomatically false
   VAR_INPUT
      Sensor_102B5 : Bool;
      Sensor_102B6 : Bool;
      Open_Valve : Bool;
   END_VAR
   VAR_OUTPUT
      Valve_106Q6 : Bool;
      Motor_4Q5 : Bool;
   END_VAR
   VAR
      Motor_Control : Bool;
   END_VAR
   VAR_TEMP   // added for the SCL form of the ladder/FBD networks
      _w1 : Bool;
   END_VAR
BEGIN

REGION Network 1
   // V 0.1.1 Updated connection for motor
   // V 0.1.0 Preliminary sketch
   // Connection for OnOff_regulator
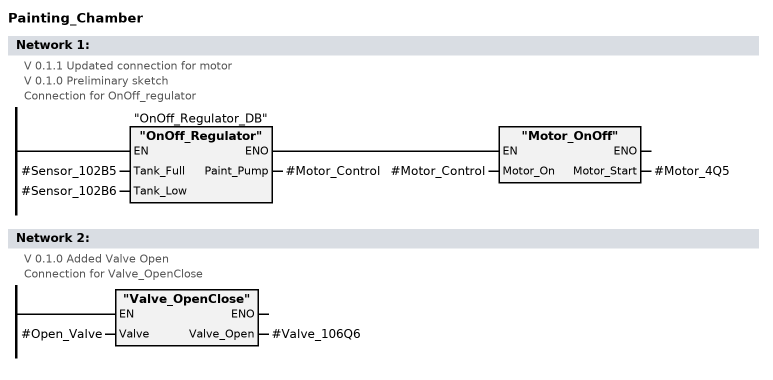
   RUNG wire#powerrail
      "OnOff_Regulator_DB"(Tank_Full := #Sensor_102B5, Tank_Low := #Sensor_102B6, Paint_Pump => #Motor_Control)
      "Motor_OnOff"(Motor_On := #Motor_Control, Motor_Start => #Motor_4Q5)
   END_RUNG
   // the same network as SCL:
   "OnOff_Regulator_DB"(Tank_Full := #Sensor_102B5,   // "OnOff_Regulator"
                        Tank_Low := #Sensor_102B6,
                        Paint_Pump => #Motor_Control,
                        ENO => #_w1);
   IF #_w1 THEN "Motor_OnOff"(Motor_On := #Motor_Control, Motor_Start => #Motor_4Q5); END_IF;
END_REGION

REGION Network 2
   // V 0.1.0 Added Valve Open
   // Connection for Valve_OpenClose
   RUNG wire#powerrail
      "Valve_OpenClose"(Valve := #Open_Valve, Valve_Open => #Valve_106Q6)
   END_RUNG
   // the same network as SCL:
   "Valve_OpenClose"(Valve := #Open_Valve, Valve_Open => #Valve_106Q6);
END_REGION
END_FUNCTION_BLOCK

FUNCTION_BLOCK "OnOff_Regulator"
{ S7_Optimized_Access := 'TRUE' }
VERSION : 0.1
   VAR_INPUT 
      Tank_Full : Bool;
      Tank_Low : Bool;
   END_VAR

   VAR_OUTPUT 
      Paint_Pump : Bool;
   END_VAR


BEGIN
	// V 0.1.0
	IF #Tank_Low=0 THEN
	    #Paint_Pump := 1;
	END_IF;
	
	IF #Tank_Full THEN
	    #Paint_Pump := 0;
	END_IF;
END_FUNCTION_BLOCK

FUNCTION "Motor_OnOff" : Void
{ S7_Optimized_Access := 'TRUE' }
VERSION : 0.1
   VAR_INPUT 
      Motor_On : Bool;
   END_VAR

   VAR_OUTPUT 
      Motor_Start : Bool;
   END_VAR


BEGIN
	IF #Motor_On THEN
	    #Motor_Start := 1;
	ELSE
	    #Motor_Start := 0;
	 
	END_IF;
	
END_FUNCTION

FUNCTION "Valve_OpenClose" : Void
{ S7_Optimized_Access := 'TRUE' }
VERSION : 0.1
   VAR_INPUT 
      Valve : Bool;
   END_VAR

   VAR_OUTPUT 
      Valve_Open : Bool;
   END_VAR


BEGIN
	IF #Valve THEN
	    #Valve_Open := 1;
	ELSE
	    #Valve_Open := 0;
	END_IF;
END_FUNCTION

FUNCTION_BLOCK "Projekt2B_RobotGrinder"   // FB1, STL
{ S7_Optimized_Access := 'TRUE' }
// stored: MemoryReserve 100
   VAR_INPUT
      Emergency_Stop_Status_150K1 : Bool;
      Sensor_102B2 : Bool;
      Sensor_102B3 : Bool;
      Sensor_102B4 : Bool;
      Sensor_102B5 : Bool;
      Sensor_102B6 : Bool;
      Reset : Bool;
   END_VAR
   VAR_OUTPUT
      Valve_106Q6 : Bool;
      Motor_4Q3 : Bool;
      Motor_4Q5 : Bool;
      Motor_6Q1 : Bool;
      Motor_6Q3 : Bool;
      Reset_Safety_150K1 : Bool;
   END_VAR
BEGIN
END_FUNCTION_BLOCK

FUNCTION_BLOCK "Storage"   // FB2, LAD
{ S7_Optimized_Access := 'TRUE' }
// V.0.1.0 - Created function block
// stored: MemoryReserve 100, SetENOAutomatically false
   VAR_INPUT
      Insert_Item : Int;   // Insert item type into storage
      Take_Item : Int;   // Remove item type from storage
      Storage_Max : Int := 5;   // Maximum storage amount allowed
      Storage_Min : Int := 3;   // Minimum storage amount after production
   END_VAR
   VAR_OUTPUT
      Storage_1 : Int;   // How many items are currently on space A
      Storage_2 : Int;   // How many items are currently on space B
      Storage_3 : Int;   // How many items are currently on space C
   END_VAR
   VAR
      Items_On_Space_1 : Int;   // Amount of items on space 1
      Items_On_Space_2 : Int;   // Amount of items on space 2
      Items_On_Space_3 : Int;   // Amount of items on space 3
   END_VAR
BEGIN

REGION Network 1: Insert items into storage
   // If inserting type X, then check if capacity is reached. If below full capacity then add item
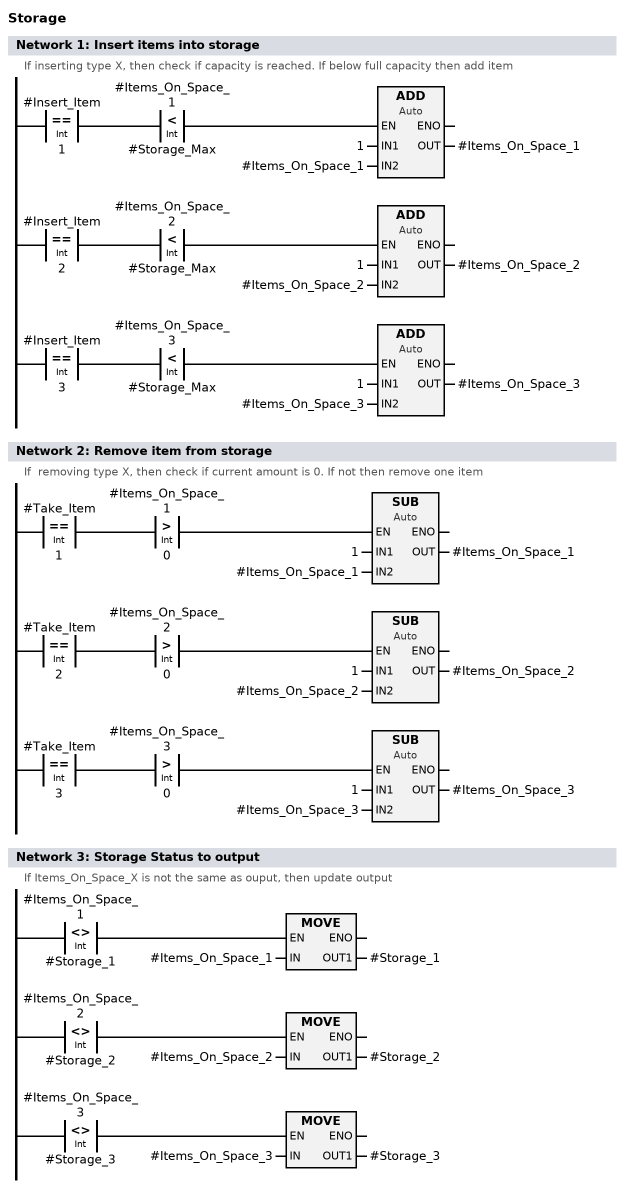
   RUNG wire#powerrail
      { S7_Templates := "SrcType := Int" } EQ_Contact(in1 := #Insert_Item, in2 := 1)
      { S7_Templates := "SrcType := Int" } LT_Contact(in1 := #Items_On_Space_1, in2 := #Storage_Max)
      Add(in1 := 1, in2 := #Items_On_Space_1, out => #Items_On_Space_1)
   END_RUNG
   RUNG wire#powerrail
      { S7_Templates := "SrcType := Int" } EQ_Contact(in1 := #Insert_Item, in2 := 2)
      { S7_Templates := "SrcType := Int" } LT_Contact(in1 := #Items_On_Space_2, in2 := #Storage_Max)
      Add(in1 := 1, in2 := #Items_On_Space_2, out => #Items_On_Space_2)
   END_RUNG
   RUNG wire#powerrail
      { S7_Templates := "SrcType := Int" } EQ_Contact(in1 := #Insert_Item, in2 := 3)
      { S7_Templates := "SrcType := Int" } LT_Contact(in1 := #Items_On_Space_3, in2 := #Storage_Max)
      Add(in1 := 1, in2 := #Items_On_Space_3, out => #Items_On_Space_3)
   END_RUNG
   // the same network as SCL:
   IF (#Insert_Item = 1) AND (#Items_On_Space_1 < #Storage_Max) THEN
       #Items_On_Space_1 := 1 + #Items_On_Space_1;
   END_IF;
   IF (#Insert_Item = 2) AND (#Items_On_Space_2 < #Storage_Max) THEN
       #Items_On_Space_2 := 1 + #Items_On_Space_2;
   END_IF;
   IF (#Insert_Item = 3) AND (#Items_On_Space_3 < #Storage_Max) THEN
       #Items_On_Space_3 := 1 + #Items_On_Space_3;
   END_IF;
END_REGION

REGION Network 2: Remove item from storage
   // If  removing type X, then check if current amount is 0. If not then remove one item
   RUNG wire#powerrail
      { S7_Templates := "SrcType := Int" } EQ_Contact(in1 := #Take_Item, in2 := 1)
      { S7_Templates := "SrcType := Int" } GT_Contact(in1 := #Items_On_Space_1, in2 := 0)
      Sub(in1 := 1, in2 := #Items_On_Space_1, out => #Items_On_Space_1)
   END_RUNG
   RUNG wire#powerrail
      { S7_Templates := "SrcType := Int" } EQ_Contact(in1 := #Take_Item, in2 := 2)
      { S7_Templates := "SrcType := Int" } GT_Contact(in1 := #Items_On_Space_2, in2 := 0)
      Sub(in1 := 1, in2 := #Items_On_Space_2, out => #Items_On_Space_2)
   END_RUNG
   RUNG wire#powerrail
      { S7_Templates := "SrcType := Int" } EQ_Contact(in1 := #Take_Item, in2 := 3)
      { S7_Templates := "SrcType := Int" } GT_Contact(in1 := #Items_On_Space_3, in2 := 0)
      Sub(in1 := 1, in2 := #Items_On_Space_3, out => #Items_On_Space_3)
   END_RUNG
   // the same network as SCL:
   IF (#Take_Item = 1) AND (#Items_On_Space_1 > 0) THEN #Items_On_Space_1 := 1 - #Items_On_Space_1; END_IF;
   IF (#Take_Item = 2) AND (#Items_On_Space_2 > 0) THEN #Items_On_Space_2 := 1 - #Items_On_Space_2; END_IF;
   IF (#Take_Item = 3) AND (#Items_On_Space_3 > 0) THEN #Items_On_Space_3 := 1 - #Items_On_Space_3; END_IF;
END_REGION

REGION Network 3: Storage Status to output
   // If Items_On_Space_X is not the same as ouput, then update output
   RUNG wire#powerrail
      { S7_Templates := "SrcType := Int" } NE_Contact(in1 := #Items_On_Space_1, in2 := #Storage_1)
      Move(in := #Items_On_Space_1, out1 => #Storage_1)
   END_RUNG
   RUNG wire#powerrail
      { S7_Templates := "SrcType := Int" } NE_Contact(in1 := #Items_On_Space_2, in2 := #Storage_2)
      Move(in := #Items_On_Space_2, out1 => #Storage_2)
   END_RUNG
   RUNG wire#powerrail
      { S7_Templates := "SrcType := Int" } NE_Contact(in1 := #Items_On_Space_3, in2 := #Storage_3)
      Move(in := #Items_On_Space_3, out1 => #Storage_3)
   END_RUNG
   // the same network as SCL:
   IF #Items_On_Space_1 <> #Storage_1 THEN #Storage_1 := #Items_On_Space_1; END_IF;
   IF #Items_On_Space_2 <> #Storage_2 THEN #Storage_2 := #Items_On_Space_2; END_IF;
   IF #Items_On_Space_3 <> #Storage_3 THEN #Storage_3 := #Items_On_Space_3; END_IF;
END_REGION
END_FUNCTION_BLOCK

FUNCTION_BLOCK "Pause"
{ S7_Optimized_Access := 'TRUE' }
VERSION : 0.1
   VAR_INPUT 
      Pause : Bool;
   END_VAR

   VAR_OUTPUT 
      Pause_Process : Bool;
   END_VAR


BEGIN
	//V0.1.0 - Created pause function
	
	IF #Pause THEN
	    #Pause_Process := 1;
	END_IF;
	
	IF #Pause AND #Pause_Process THEN
	    #Pause_Process := 0;
	END_IF;
	
END_FUNCTION_BLOCK

FUNCTION "Teeeeeeeeest" : Void
{ S7_Optimized_Access := 'TRUE' }
VERSION : 0.1

BEGIN
END_FUNCTION

FUNCTION_BLOCK "Test_Function_Block"
{ S7_Optimized_Access := 'TRUE' }
VERSION : 0.1

BEGIN
	// Kan i se det her??
END_FUNCTION_BLOCK

FUNCTION "conveyor_belt_Back_And_Forth" : Void
{ S7_Optimized_Access := 'TRUE' }
VERSION : 0.1
   VAR_INPUT 
      Input_conveyor_belt_forward : Bool;
      Input_conveyor_belt_back : Bool;
   END_VAR

   VAR_OUTPUT 
      "Output_Conveyor Belt Forward" : Bool;
      "Output_Conveyor Belt Back" : Bool;
      "Output_Conveyor Belt Ready" : Bool;
   END_VAR


BEGIN
	//V0.0.1 
	
	#"Output_Conveyor Belt Forward" := 0;
	#"Output_Conveyor Belt Back" := 0;
	#"Output_Conveyor Belt Ready" := 0;
	
	IF #Input_conveyor_belt_forward THEN
	    #"Output_Conveyor Belt Forward" := 1;
	    #"Output_Conveyor Belt Ready" := 1;
	ELSIF #Input_conveyor_belt_back THEN
	    #"Output_Conveyor Belt Back" := 1;
	    #"Output_Conveyor Belt Ready" := 1;
	END_IF;
	
END_FUNCTION

DATA_BLOCK "FC_Modbus_Arduino_DB"   // DB4
// stored: InstanceOfName FC_Modbus_Arduino, InstanceOfType FB
"FC_Modbus_Arduino"
BEGIN
END_DATA_BLOCK

DATA_BLOCK "MB_CLIENT_DB_Arduino_Read"   // DB1
// stored: InstanceOfName MB_CLIENT, OfSystemLibElement MB_CLIENT, OfSystemLibVersion 6.0
"MB_CLIENT"
   // VAR_INPUT
   //    REQ : Bool;
   //    DISCONNECT : Bool;
   //    MB_MODE : USInt;
   //    MB_DATA_ADDR : UDInt;
   //    MB_DATA_LEN : UInt;
   //    RD_MB_DATA_ADDR : UInt;
   //    RD_MB_DATA_LEN : UInt;
   //    WR_MB_DATA_ADDR : UInt;
   //    WR_MB_DATA_LEN : UInt;
   // END_VAR
   // VAR_OUTPUT
   //    DONE : Bool;
   //    BUSY : Bool;
   //    ERROR : Bool;
   //    STATUS { ExternalVisible := 'False'} : Word;
   // END_VAR
   // VAR_IN_OUT
   //    MB_DATA_PTR : Variant;
   //    CONNECT : Variant;
   //    RD_MB_DATA_PTR : Variant;
   //    WR_MB_DATA_PTR : Variant;
   // END_VAR
   // VAR
   //    TCON { S7_SetPoint := 'True'} : TCON;
   //    TDISCON { S7_SetPoint := 'True'} : TDISCON;
   //    TSEND { S7_SetPoint := 'True'} : TSEND;
   //    TRECEIVE { S7_SetPoint := 'True'} : TRCV;
   //    TRESET { S7_SetPoint := 'True'} : T_RESET;
   //    TDIAG { S7_SetPoint := 'True'} : T_DIAG;
   //    TDIAG_Status { S7_SetPoint := 'True'} : TDiag_Status;
   //    Blocked_Proc_Timeout : Real;
   //    Rcv_Timeout : Real;
   //    MB_Unit_ID : Byte;
   //    MB_Transaction_ID : Word;
   //    RD_MB_DATA_PTR_Length : UDInt;
   //    WR_MB_DATA_PTR_Length : UDInt;
   //    MB_State { ExternalWritable := 'False'} : Word;
   //    SAVED_MB_DATA_ADDR : UDInt;
   //    SAVED_DATA_LEN : UInt;
   //    SAVED_MB_MODE : USInt;
   //    Connection_ID : Word;
   //    Retries : Word;
   //    TEMP_DATA { ExternalWritable := 'False'} : Array[1..263] of Byte;
   //    rcv_timer { ExternalAccessible := 'False'; ExternalVisible := 'False'; ExternalWritable := 'False'; S7_SetPoint := 'True'} : TON_TIME;
   //    wd_timer { ExternalAccessible := 'False'; ExternalVisible := 'False'; ExternalWritable := 'False'; S7_SetPoint := 'True'} : TON_TIME;
   //    Connected : Bool;
   //    Active { ExternalWritable := 'False'} : Bool;
   //    BytesReceived : UDInt;
   //    Func_Code_23_saved { ExternalAccessible := 'False'; ExternalVisible := 'False'; ExternalWritable := 'False'} : Struct
   //       mb_data_addr_read : Word;
   //       mb_data_len_read : Word;
   //       mb_data_addr_write : Word;
   //       mb_data_len_write : Word;
   //    END_STRUCT;
   // END_VAR
BEGIN
END_DATA_BLOCK

DATA_BLOCK "MB_CLIENT_DB_Arduino_Write"   // DB13
// stored: InstanceOfName MB_CLIENT, OfSystemLibElement MB_CLIENT, OfSystemLibVersion 6.0
"MB_CLIENT"
   // VAR_INPUT
   //    REQ : Bool;
   //    DISCONNECT : Bool;
   //    MB_MODE : USInt;
   //    MB_DATA_ADDR : UDInt;
   //    MB_DATA_LEN : UInt;
   //    RD_MB_DATA_ADDR : UInt;
   //    RD_MB_DATA_LEN : UInt;
   //    WR_MB_DATA_ADDR : UInt;
   //    WR_MB_DATA_LEN : UInt;
   // END_VAR
   // VAR_OUTPUT
   //    DONE : Bool;
   //    BUSY : Bool;
   //    ERROR : Bool;
   //    STATUS { ExternalVisible := 'False'} : Word;
   // END_VAR
   // VAR_IN_OUT
   //    MB_DATA_PTR : Variant;
   //    CONNECT : Variant;
   //    RD_MB_DATA_PTR : Variant;
   //    WR_MB_DATA_PTR : Variant;
   // END_VAR
   // VAR
   //    TCON { S7_SetPoint := 'True'} : TCON;
   //    TDISCON { S7_SetPoint := 'True'} : TDISCON;
   //    TSEND { S7_SetPoint := 'True'} : TSEND;
   //    TRECEIVE { S7_SetPoint := 'True'} : TRCV;
   //    TRESET { S7_SetPoint := 'True'} : T_RESET;
   //    TDIAG { S7_SetPoint := 'True'} : T_DIAG;
   //    TDIAG_Status { S7_SetPoint := 'True'} : TDiag_Status;
   //    Blocked_Proc_Timeout : Real;
   //    Rcv_Timeout : Real;
   //    MB_Unit_ID : Byte;
   //    MB_Transaction_ID : Word;
   //    RD_MB_DATA_PTR_Length : UDInt;
   //    WR_MB_DATA_PTR_Length : UDInt;
   //    MB_State { ExternalWritable := 'False'} : Word;
   //    SAVED_MB_DATA_ADDR : UDInt;
   //    SAVED_DATA_LEN : UInt;
   //    SAVED_MB_MODE : USInt;
   //    Connection_ID : Word;
   //    Retries : Word;
   //    TEMP_DATA { ExternalWritable := 'False'} : Array[1..263] of Byte;
   //    rcv_timer { ExternalAccessible := 'False'; ExternalVisible := 'False'; ExternalWritable := 'False'; S7_SetPoint := 'True'} : TON_TIME;
   //    wd_timer { ExternalAccessible := 'False'; ExternalVisible := 'False'; ExternalWritable := 'False'; S7_SetPoint := 'True'} : TON_TIME;
   //    Connected : Bool;
   //    Active { ExternalWritable := 'False'} : Bool;
   //    BytesReceived : UDInt;
   //    Func_Code_23_saved { ExternalAccessible := 'False'; ExternalVisible := 'False'; ExternalWritable := 'False'} : Struct
   //       mb_data_addr_read : Word;
   //       mb_data_len_read : Word;
   //       mb_data_addr_write : Word;
   //       mb_data_len_write : Word;
   //    END_STRUCT;
   // END_VAR
BEGIN
END_DATA_BLOCK

DATA_BLOCK "Projekt2B_RobotGrinder_DB"   // DB1
// stored: InstanceOfName Projekt2B_RobotGrinder, InstanceOfType FB
"Projekt2B_RobotGrinder"
BEGIN
END_DATA_BLOCK

DATA_BLOCK "Projekt_2B_Robotgrinder_DB"   // DB1
// stored: InstanceOfName Projekt_2B_Robotgrinder, InstanceOfType FB
"Projekt_2B_Robotgrinder"
BEGIN
END_DATA_BLOCK

DATA_BLOCK "Robot_Modbus_DB"   // DB1
// stored: InstanceOfName Robot_Modbus, InstanceOfType FB
"Robot_Modbus"
BEGIN
END_DATA_BLOCK

DATA_BLOCK "Timer_Paint"   // DB6
{ S7_Optimized_Access := 'TRUE' }
// stored: InstanceOfName IEC_TIMER, OfSystemLibElement IEC_TIMER, OfSystemLibVersion 1.0
"IEC_TIMER"
   // VAR
   //    PT : Time;
   //    ET { ExternalWritable := 'False'} : Time;
   //    IN : Bool;
   //    Q { ExternalWritable := 'False'} : Bool;
   // END_VAR
BEGIN
END_DATA_BLOCK

DATA_BLOCK "Modbus_Coordinates"   // DB4
// stored: InstanceOfName MB_CLIENT, OfSystemLibElement MB_CLIENT, OfSystemLibVersion 6.0
"MB_CLIENT"
   // VAR_INPUT
   //    REQ : Bool;
   //    DISCONNECT : Bool;
   //    MB_MODE : USInt;
   //    MB_DATA_ADDR : UDInt;
   //    MB_DATA_LEN : UInt;
   //    RD_MB_DATA_ADDR : UInt;
   //    RD_MB_DATA_LEN : UInt;
   //    WR_MB_DATA_ADDR : UInt;
   //    WR_MB_DATA_LEN : UInt;
   // END_VAR
   // VAR_OUTPUT
   //    DONE : Bool;
   //    BUSY : Bool;
   //    ERROR : Bool;
   //    STATUS { ExternalVisible := 'False'} : Word;
   // END_VAR
   // VAR_IN_OUT
   //    MB_DATA_PTR : Variant;
   //    CONNECT : Variant;
   //    RD_MB_DATA_PTR : Variant;
   //    WR_MB_DATA_PTR : Variant;
   // END_VAR
   // VAR
   //    TCON { S7_SetPoint := 'True'} : TCON;
   //    TDISCON { S7_SetPoint := 'True'} : TDISCON;
   //    TSEND { S7_SetPoint := 'True'} : TSEND;
   //    TRECEIVE { S7_SetPoint := 'True'} : TRCV;
   //    TRESET { S7_SetPoint := 'True'} : T_RESET;
   //    TDIAG { S7_SetPoint := 'True'} : T_DIAG;
   //    TDIAG_Status { S7_SetPoint := 'True'} : TDiag_Status;
   //    Blocked_Proc_Timeout : Real;
   //    Rcv_Timeout : Real;
   //    MB_Unit_ID : Byte;
   //    MB_Transaction_ID : Word;
   //    RD_MB_DATA_PTR_Length : UDInt;
   //    WR_MB_DATA_PTR_Length : UDInt;
   //    MB_State { ExternalWritable := 'False'} : Word;
   //    SAVED_MB_DATA_ADDR : UDInt;
   //    SAVED_DATA_LEN : UInt;
   //    SAVED_MB_MODE : USInt;
   //    Connection_ID : Word;
   //    Retries : Word;
   //    TEMP_DATA { ExternalWritable := 'False'} : Array[1..263] of Byte;
   //    rcv_timer { ExternalAccessible := 'False'; ExternalVisible := 'False'; ExternalWritable := 'False'; S7_SetPoint := 'True'} : TON_TIME;
   //    wd_timer { ExternalAccessible := 'False'; ExternalVisible := 'False'; ExternalWritable := 'False'; S7_SetPoint := 'True'} : TON_TIME;
   //    Connected : Bool;
   //    Active { ExternalWritable := 'False'} : Bool;
   //    BytesReceived : UDInt;
   //    Func_Code_23_saved { ExternalAccessible := 'False'; ExternalVisible := 'False'; ExternalWritable := 'False'} : Struct
   //       mb_data_addr_read : Word;
   //       mb_data_len_read : Word;
   //       mb_data_addr_write : Word;
   //       mb_data_len_write : Word;
   //    END_STRUCT;
   // END_VAR
BEGIN
END_DATA_BLOCK

DATA_BLOCK "Modbus_Receive"   // DB2
// stored: InstanceOfName MB_CLIENT, OfSystemLibElement MB_CLIENT, OfSystemLibVersion 6.0
"MB_CLIENT"
   // VAR_INPUT
   //    REQ : Bool;
   //    DISCONNECT : Bool;
   //    MB_MODE : USInt;
   //    MB_DATA_ADDR : UDInt;
   //    MB_DATA_LEN : UInt;
   //    RD_MB_DATA_ADDR : UInt;
   //    RD_MB_DATA_LEN : UInt;
   //    WR_MB_DATA_ADDR : UInt;
   //    WR_MB_DATA_LEN : UInt;
   // END_VAR
   // VAR_OUTPUT
   //    DONE : Bool;
   //    BUSY : Bool;
   //    ERROR : Bool;
   //    STATUS { ExternalVisible := 'False'} : Word;
   // END_VAR
   // VAR_IN_OUT
   //    MB_DATA_PTR : Variant;
   //    CONNECT : Variant;
   //    RD_MB_DATA_PTR : Variant;
   //    WR_MB_DATA_PTR : Variant;
   // END_VAR
   // VAR
   //    TCON { S7_SetPoint := 'True'} : TCON;
   //    TDISCON { S7_SetPoint := 'True'} : TDISCON;
   //    TSEND { S7_SetPoint := 'True'} : TSEND;
   //    TRECEIVE { S7_SetPoint := 'True'} : TRCV;
   //    TRESET { S7_SetPoint := 'True'} : T_RESET;
   //    TDIAG { S7_SetPoint := 'True'} : T_DIAG;
   //    TDIAG_Status { S7_SetPoint := 'True'} : TDiag_Status;
   //    Blocked_Proc_Timeout : Real;
   //    Rcv_Timeout : Real;
   //    MB_Unit_ID : Byte;
   //    MB_Transaction_ID : Word;
   //    RD_MB_DATA_PTR_Length : UDInt;
   //    WR_MB_DATA_PTR_Length : UDInt;
   //    MB_State { ExternalWritable := 'False'} : Word;
   //    SAVED_MB_DATA_ADDR : UDInt;
   //    SAVED_DATA_LEN : UInt;
   //    SAVED_MB_MODE : USInt;
   //    Connection_ID : Word;
   //    Retries : Word;
   //    TEMP_DATA { ExternalWritable := 'False'} : Array[1..263] of Byte;
   //    rcv_timer { ExternalAccessible := 'False'; ExternalVisible := 'False'; ExternalWritable := 'False'; S7_SetPoint := 'True'} : TON_TIME;
   //    wd_timer { ExternalAccessible := 'False'; ExternalVisible := 'False'; ExternalWritable := 'False'; S7_SetPoint := 'True'} : TON_TIME;
   //    Connected : Bool;
   //    Active { ExternalWritable := 'False'} : Bool;
   //    BytesReceived : UDInt;
   //    Func_Code_23_saved { ExternalAccessible := 'False'; ExternalVisible := 'False'; ExternalWritable := 'False'} : Struct
   //       mb_data_addr_read : Word;
   //       mb_data_len_read : Word;
   //       mb_data_addr_write : Word;
   //       mb_data_len_write : Word;
   //    END_STRUCT;
   // END_VAR
BEGIN
END_DATA_BLOCK

DATA_BLOCK "Modbus_Write"   // DB3
// stored: InstanceOfName MB_CLIENT, OfSystemLibElement MB_CLIENT, OfSystemLibVersion 6.0
"MB_CLIENT"
   // VAR_INPUT
   //    REQ : Bool;
   //    DISCONNECT : Bool;
   //    MB_MODE : USInt;
   //    MB_DATA_ADDR : UDInt;
   //    MB_DATA_LEN : UInt;
   //    RD_MB_DATA_ADDR : UInt;
   //    RD_MB_DATA_LEN : UInt;
   //    WR_MB_DATA_ADDR : UInt;
   //    WR_MB_DATA_LEN : UInt;
   // END_VAR
   // VAR_OUTPUT
   //    DONE : Bool;
   //    BUSY : Bool;
   //    ERROR : Bool;
   //    STATUS { ExternalVisible := 'False'} : Word;
   // END_VAR
   // VAR_IN_OUT
   //    MB_DATA_PTR : Variant;
   //    CONNECT : Variant;
   //    RD_MB_DATA_PTR : Variant;
   //    WR_MB_DATA_PTR : Variant;
   // END_VAR
   // VAR
   //    TCON { S7_SetPoint := 'True'} : TCON;
   //    TDISCON { S7_SetPoint := 'True'} : TDISCON;
   //    TSEND { S7_SetPoint := 'True'} : TSEND;
   //    TRECEIVE { S7_SetPoint := 'True'} : TRCV;
   //    TRESET { S7_SetPoint := 'True'} : T_RESET;
   //    TDIAG { S7_SetPoint := 'True'} : T_DIAG;
   //    TDIAG_Status { S7_SetPoint := 'True'} : TDiag_Status;
   //    Blocked_Proc_Timeout : Real;
   //    Rcv_Timeout : Real;
   //    MB_Unit_ID : Byte;
   //    MB_Transaction_ID : Word;
   //    RD_MB_DATA_PTR_Length : UDInt;
   //    WR_MB_DATA_PTR_Length : UDInt;
   //    MB_State { ExternalWritable := 'False'} : Word;
   //    SAVED_MB_DATA_ADDR : UDInt;
   //    SAVED_DATA_LEN : UInt;
   //    SAVED_MB_MODE : USInt;
   //    Connection_ID : Word;
   //    Retries : Word;
   //    TEMP_DATA { ExternalWritable := 'False'} : Array[1..263] of Byte;
   //    rcv_timer { ExternalAccessible := 'False'; ExternalVisible := 'False'; ExternalWritable := 'False'; S7_SetPoint := 'True'} : TON_TIME;
   //    wd_timer { ExternalAccessible := 'False'; ExternalVisible := 'False'; ExternalWritable := 'False'; S7_SetPoint := 'True'} : TON_TIME;
   //    Connected : Bool;
   //    Active { ExternalWritable := 'False'} : Bool;
   //    BytesReceived : UDInt;
   //    Func_Code_23_saved { ExternalAccessible := 'False'; ExternalVisible := 'False'; ExternalWritable := 'False'} : Struct
   //       mb_data_addr_read : Word;
   //       mb_data_len_read : Word;
   //       mb_data_addr_write : Word;
   //       mb_data_len_write : Word;
   //    END_STRUCT;
   // END_VAR
BEGIN
END_DATA_BLOCK

DATA_BLOCK "Robot_Working_Oneshot"   // DB8
// stored: InstanceOfName R_TRIG, OfSystemLibElement R_TRIG, OfSystemLibVersion 1.0
"R_TRIG"
   // VAR_INPUT
   //    CLK : Bool;
   // END_VAR
   // VAR_OUTPUT
   //    Q : Bool;
   // END_VAR
   // VAR
   //    Stat_Bit : Bool;
   // END_VAR
BEGIN
END_DATA_BLOCK
